{attribute addProperty BoxType "EK1100-0000-0018"}
{attribute addProperty Id "Beckhoff_AX5xxxEK1122Beckhoff_AX5xxxEK1122_5EFAAD43586707333.75"}
{attribute addProperty CRC "2879638353"}
{attribute addProperty SizeInBites "58670"}
{attribute addProperty SizeInBytes "7333.75"}
TYPE Beckhoff_AX5xxx_ABA3CB51 EXTENDS EK1100_179A0949 :
STRUCT
	{attribute addProperty Name "Beckhoff_AX5xxxEK1122"}
	Beckhoff_AX5xxxEK1122 : Beckhoff_AX5xxxEK1122_5EFAAD43;
END_STRUCT
END_TYPE

(* stored: Version 1.2.0.0, ProductVersion 3.1.4024.9
   DUT Beckhoff_AX5xxx_ABA3CB51: Id {85ddbeda-b3a1-4d82-abca-0e217503c24b} *)
